Fanuc KAREL source: ka00066.KL

PROGRAM KA00066
%NOLOCKGROUP
VAR
SRC : XYZWPR;DST : XYZWPR
BEGIN
--
SRC.X=1.0
DST=SRC
END KA00066
